FUNCTION_BLOCK FB_AO EXTENDS FB_Basic
VAR_INPUT
	rValue		: LREAL;
END_VAR
VAR_OUTPUT
END_VAR
VAR
	fbLinTrafo	: FB_LIN_TRAFO;

// HW
	{attribute 'OPC.UA.DA':='1'}
	{attribute 'OPC.UA.DA.Access' := '1'}
	{attribute 'OPC.UA.DA.Description' := 'Output I/O signal (RAW)'}
	{attribute 'OPC.UA.DA.StructuredType' := '0'}
	AnalogOutput AT %Q* : INT;	// Value to IO module
	State AT %I* : UINT := 8;	// State from Ethercat module
	AdsAdrr AT %I* : AMSADDR;	// ADS address from EtherCAT module

END_VAR
VAR PERSISTENT
	rScaleMax	: LREAL := 100;
	rScaleMin	: LREAL := -100;

END_VAR


// Run parent FB
SUPER^();

METHOD PROTECTED M_AutoMode : BOOL
VAR_INPUT
END_VAR
// Analog output automatic mode
// Executed from parent FB_Basic

rAutoValue := rValue;

IF (P_bEnable) THEN
	rActualValue := rAutoValue;
ELSE
	rActualValue := 0.0;
END_IF
END_METHOD

METHOD PROTECTED M_ErrorHandling : BOOL
VAR_INPUT
END_VAR
// Error handling
IF (bCmdEnable) THEN
	IF (NOT P_bManualMode) THEN
		// Hardware errors
		IF (NOT F_ECat_OK(State)) THEN
			// EtherCAT state
			bStaError := TRUE;
			eStaErrorID := E_ComponentErrors.HW_ECat_Not_OP;
		END_IF
	END_IF
	
ELSE
	bStaError := FALSE;
	bStaWarning := FALSE;
	eStaErrorID := E_ComponentErrors.OK;

END_IF
END_METHOD

METHOD PROTECTED M_Init : BOOL
VAR_INPUT
END_VAR
// Init

bCmdEnable := TRUE;
bInitDone := TRUE;
END_METHOD

METHOD PROTECTED M_ManualMode : BOOL
VAR_INPUT
END_VAR
// Analog Output manual mode
// Executed from parent FB_Basic

rManualValue := LIMIT(rScaleMin, rManualValue, rScaleMax);

IF (P_bEnable) THEN
	rActualValue := rManualValue;
ELSE
	rActualValue := 0.0;
END_IF
END_METHOD

METHOD PROTECTED M_Run : BOOL
VAR_INPUT
END_VAR
// Analog outputs run
// Executed from parent FB_Basic

// Update IO 

fbLinTrafo(	rIN := rActualValue,
			rIN_MIN := rScaleMin,
			rIN_MAX := rScaleMax,
			rOUT_MIN := -32767,
			rOUT_MAX := 32767,
			rOUT => ,
			bERROR =>	);

AnalogOutput := LREAL_TO_INT(fbLinTrafo.rOUT);
END_METHOD

PROPERTY PUBLIC P_rScaleMax : LREAL
GET
P_rScaleMax := rScaleMax;
END_GET
SET
rScaleMax := P_rScaleMax;
END_SET
END_PROPERTY

PROPERTY PUBLIC P_rScaleMin : LREAL
GET
P_rScaleMin := rScaleMin;
END_GET
SET
rScaleMin := P_rScaleMin;
END_SET
END_PROPERTY

END_FUNCTION_BLOCK

(* stored: Version 1.1.0.1, ProductVersion 3.1.4024.2
   POU FB_AO: Id {9fa16736-27ea-49ed-9af0-0ab83936e0b7}, SpecialFunc None
   Method M_AutoMode: Id {f245e704-90a3-4179-bdbf-fea1e18317d9}
   Method M_ErrorHandling: Id {b90a5d88-3655-4424-b22a-6f9fbf89bc41}
   Method M_Init: Id {c1fbf982-fcb3-4fe8-9448-51448a4266ec}
   Method M_ManualMode: Id {01072cf1-5ded-4d0c-87a3-457c4656934d}
   Method M_Run: Id {cb71e432-a3f6-4619-8861-41ef5909bb16}
   Property P_rScaleMax: Id {626bd2db-faa4-488f-82cf-def3763b97dd}
   Get Get: Id {8e58ad9b-f723-4e56-82f6-a6e6a191ed94}
   Set Set: Id {38490acd-4738-4c83-91f3-a2f0f15f59ce}
   Property P_rScaleMin: Id {223a6fcb-d15f-4664-b482-5b8e05776893}
   Get Get: Id {271fe616-64ef-4a2e-8ca1-53279acbf0be}
   Set Set: Id {0e13791c-87cf-4dd5-94ce-e54323023eb1} *)
